FUNCTION_BLOCK FB_EventLogger

VAR
	aEventBuffer: ARRAY[1..100] OF ST_Event;
	CurrentEventBufferIndex : INT :=0;
	_PersistentEventStorage : I_PersistentEventStorage;
END_VAR

VAR CONSTANT
     MAX_SIZE_OF_EVENT_BUFFER : INT := 100;
END_VAR

(* Return true if add was successfull and FALSE if buffer is full *)

METHOD AddEvent : BOOL
VAR_INPUT
	eEventType : E_EventType;
	eEventSeverity : TcEventSeverity;
	nEventIdentity : UDINT;
	sEventText : STRING(255);
END_VAR
IF NOT isEventBufferFull() THEN 
	CurrentEventBufferIndex := CurrentEventBufferIndex +1;
	aEventBuffer[CurrentEventBufferIndex].eEventType := eEventType;
	aEventBuffer[CurrentEventBufferIndex].eEventSeverity := eEventSeverity;
	aEventBuffer[CurrentEventBufferIndex].nEventIdentity := nEventIdentity;
	aEventBuffer[CurrentEventBufferIndex].sEventText := sEventText;
	F_UpdateEventTimeStamp(stEvent := aEventBuffer[CurrentEventBufferIndex]);
	AddEvent := TRUE;
ELSE
    AddEvent := FALSE;
END_IF


// Here we want to store the event the store Persistently
_PersistentEventStorage.StoreEvent(stEvent := aEventBuffer[CurrentEventBufferIndex]);
END_METHOD

METHOD FB_init : BOOL
VAR_INPUT
	bInitRetains : BOOL; // if TRUE, the retain variables are initialized (warm start / cold start)
	bInCopyCode : BOOL;  // if TRUE, the instance afterwards gets moved into the copy code (online change)
    iPersistentEventStorage : I_PersistentEventStorage;
END_VAR
_PersistentEventStorage := iPersistentEventStorage ;
END_METHOD

METHOD PRIVATE IsEventBufferFull : BOOL
VAR_INPUT
END_VAR
IF (CurrentEventBufferIndex + 1) > MAX_SIZE_OF_EVENT_BUFFER THEN
	isEventBufferFull := TRUE;
ELSE
		isEventBufferFull  := FALSE;
END_IF
END_METHOD

END_FUNCTION_BLOCK

(* stored: Version 1.1.0.1, ProductVersion 3.1.4024.16
   POU FB_EventLogger: Id {713a3acf-30a9-4e9b-9e75-d8979738a9f1}, SpecialFunc None
   Method AddEvent: Id {b04487a2-b847-4f72-afc1-877684e951b9}
   Method FB_init: Id {8b5a3fcd-36ea-4e7d-aee0-ef9ce3bf1017}
   Method IsEventBufferFull: Id {da0c0439-1203-4afa-a6e8-36ce13cfb0d1} *)
